TYPE ST_BasicCommand :
STRUCT
	stCmd		: ST_CommandControl;
END_STRUCT
END_TYPE

(* stored: Version 1.1.0.1, ProductVersion 3.1.4022.9
   DUT ST_BasicCommand: Id {e852155f-a12c-4f3a-a110-629ca4aa8259} *)
